FUNCTION_BLOCK FlushingManagerEffluent (* Basic Function Block Type *)
  (* Standard: 61499-2 *)
  (* Version 0.0, 8/23/2024, SESA713705, Schneider Electric, Template *)
  PACKAGE SE.Nereda;
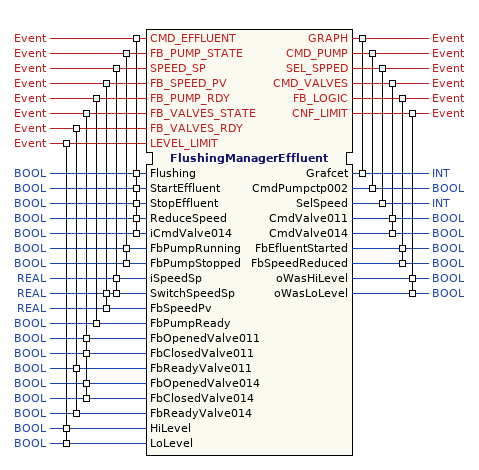
  EVENT_INPUT
    CMD_EFFLUENT WITH StartEffluent, StopEffluent, ReduceSpeed, iCmdValve014, Flushing;
    FB_PUMP_STATE WITH FbPumpRunning, FbPumpStopped;
    SPEED_SP WITH SwitchSpeedSp, iSpeedSp;
    FB_SPEED_PV WITH FbSpeedPv, SwitchSpeedSp;
    FB_PUMP_RDY WITH FbPumpReady;
    FB_VALVES_STATE WITH FbOpenedValve014, FbClosedValve014, FbOpenedValve011, FbClosedValve011;
    FB_VALVES_RDY WITH FbReadyValve011, FbReadyValve014;
    LEVEL_LIMIT WITH HiLevel, LoLevel;
  END_EVENT
  EVENT_OUTPUT
    GRAPH WITH Grafcet;
    CMD_PUMP WITH CmdPumpctp002;
    SEL_SPPED WITH SelSpeed;
    CMD_VALVES WITH CmdValve011, CmdValve014;
    FB_LOGIC WITH FbEfluentStarted, FbSpeedReduced;
    CNF_LIMIT WITH oWasHiLevel, oWasLoLevel;
  END_EVENT
  VAR_INPUT
    Flushing : BOOL;
    StartEffluent : BOOL;
    StopEffluent : BOOL;
    ReduceSpeed : BOOL;
    iCmdValve014 : BOOL;
    FbPumpRunning : BOOL;
    FbPumpStopped : BOOL;
    iSpeedSp : REAL;
    SwitchSpeedSp : REAL;
    FbSpeedPv : REAL;
    FbPumpReady : BOOL;
    FbOpenedValve011 : BOOL;
    FbClosedValve011 : BOOL;
    FbReadyValve011 : BOOL;
    FbOpenedValve014 : BOOL;
    FbClosedValve014 : BOOL;
    FbReadyValve014 : BOOL;
    HiLevel : BOOL;
    LoLevel : BOOL;
  END_VAR
  VAR_OUTPUT
    Grafcet : INT;
    CmdPumpctp002 : BOOL;
    SelSpeed : INT;
    CmdValve011 : BOOL;
    CmdValve014 : BOOL;
    FbEfluentStarted : BOOL;
    FbSpeedReduced : BOOL;
    oWasHiLevel : BOOL;
    oWasLoLevel : BOOL;
  END_VAR
  VAR
    InGSInstaActive : BOOL;
    InGSsActive : BOOL;
    InSLBActive : BOOL;
    WasHiLevel : BOOL := FALSE;
    WasLoLevel : BOOL := TRUE;
  END_VAR
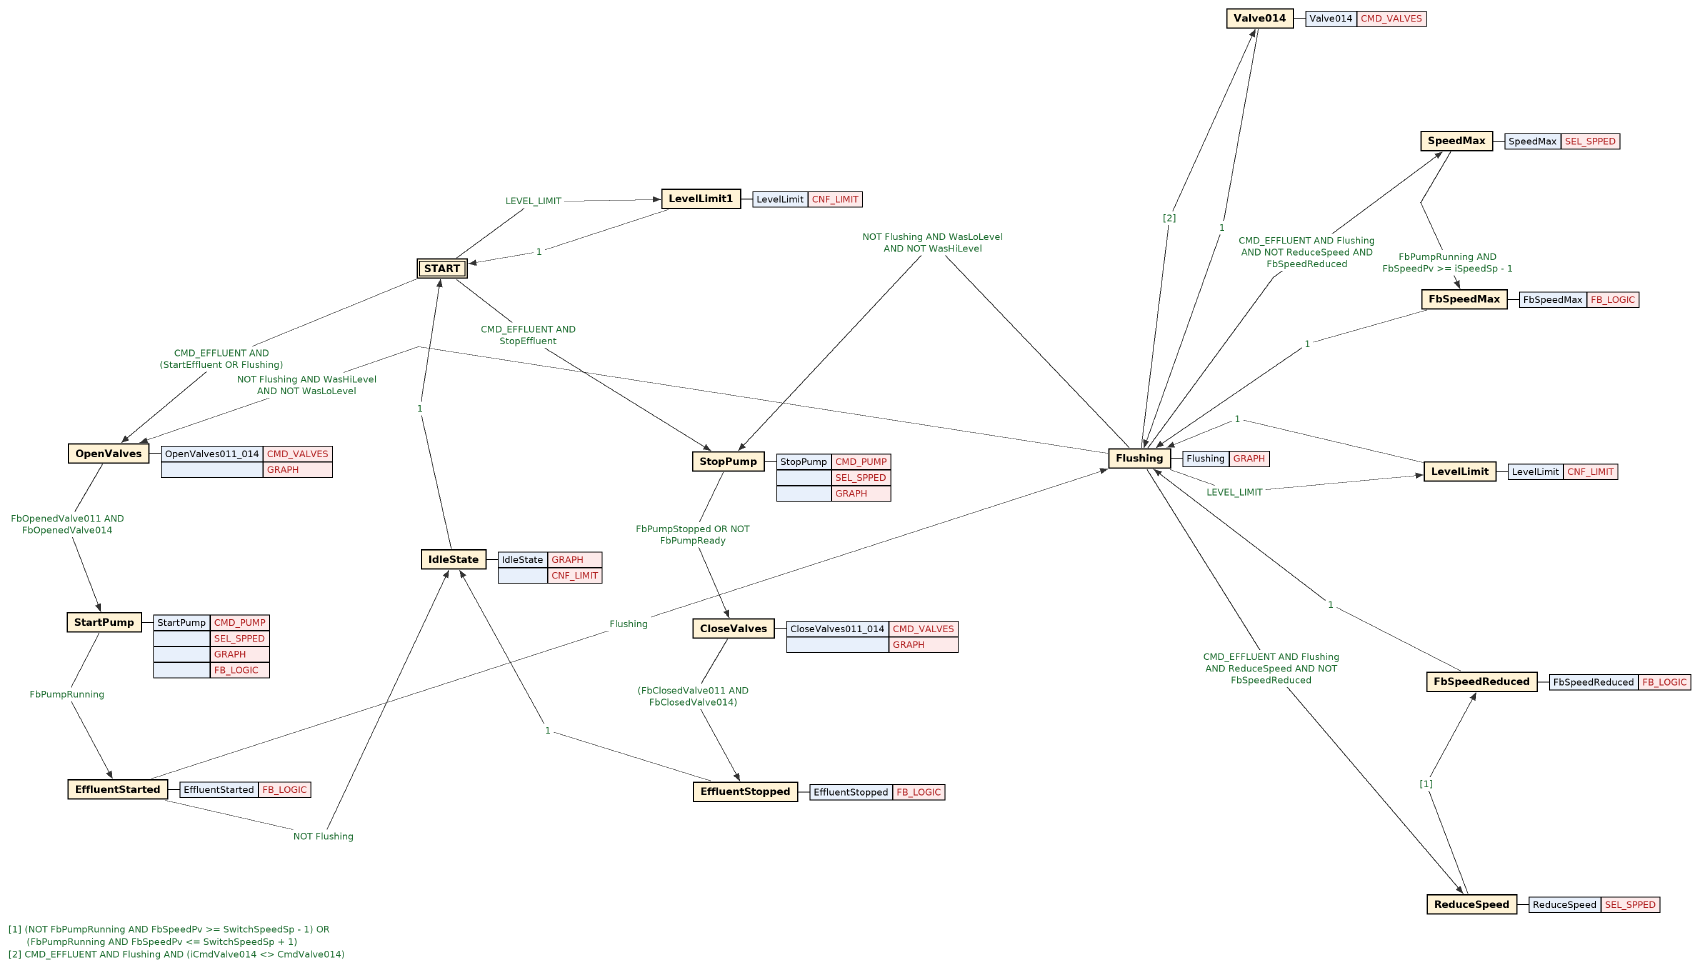
  EC_STATES
    START; (* Initial State *)
    OpenValves : OpenValves011_014 -> CMD_VALVES, -> GRAPH;
    StartPump : StartPump -> CMD_PUMP, -> SEL_SPPED, -> GRAPH, -> FB_LOGIC;
    StopPump : StopPump -> CMD_PUMP, -> SEL_SPPED, -> GRAPH;
    CloseValves : CloseValves011_014 -> CMD_VALVES, -> GRAPH;
    IdleState : IdleState -> GRAPH, -> CNF_LIMIT;
    ReduceSpeed : ReduceSpeed -> SEL_SPPED;
    SpeedMax : SpeedMax -> SEL_SPPED;
    EffluentStarted : EffluentStarted -> FB_LOGIC;
    EffluentStopped : EffluentStopped -> FB_LOGIC;
    FbSpeedMax : FbSpeedMax -> FB_LOGIC;
    FbSpeedReduced : FbSpeedReduced -> FB_LOGIC;
    Valve014 : Valve014 -> CMD_VALVES;
    Flushing : Flushing -> GRAPH;
    LevelLimit : LevelLimit -> CNF_LIMIT;
    LevelLimit1 : LevelLimit -> CNF_LIMIT;
  END_STATES
  EC_TRANSITIONS
    START TO StopPump := CMD_EFFLUENT AND StopEffluent;
    START TO OpenValves := CMD_EFFLUENT AND (StartEffluent OR Flushing);
    OpenValves TO StartPump := FbOpenedValve011 AND FbOpenedValve014;
    EffluentStarted TO IdleState := NOT Flushing;
    StopPump TO CloseValves := FbPumpStopped OR NOT FbPumpReady;
    IdleState TO START := 1;
    Flushing TO StopPump := NOT Flushing AND WasLoLevel AND NOT WasHiLevel;
    Flushing TO ReduceSpeed := CMD_EFFLUENT AND Flushing AND ReduceSpeed AND NOT FbSpeedReduced;
    FbSpeedReduced TO Flushing := 1;
    Flushing TO SpeedMax := CMD_EFFLUENT AND Flushing AND NOT ReduceSpeed AND FbSpeedReduced;
    FbSpeedMax TO Flushing := 1;
    StartPump TO EffluentStarted := FbPumpRunning;
    CloseValves TO EffluentStopped := (FbClosedValve011 AND FbClosedValve014);
    SpeedMax TO FbSpeedMax := FbPumpRunning AND FbSpeedPv >= iSpeedSp - 1;
    ReduceSpeed TO FbSpeedReduced := (NOT FbPumpRunning AND FbSpeedPv >= SwitchSpeedSp - 1) OR (FbPumpRunning AND FbSpeedPv <= SwitchSpeedSp + 1);
    Flushing TO Valve014 := CMD_EFFLUENT AND Flushing AND (iCmdValve014 <> CmdValve014);
    Valve014 TO Flushing := 1;
    EffluentStarted TO Flushing := Flushing;
    Flushing TO OpenValves := NOT Flushing AND WasHiLevel AND NOT WasLoLevel;
    Flushing TO LevelLimit := LEVEL_LIMIT;
    LevelLimit TO Flushing := 1;
    EffluentStopped TO IdleState := 1;
    START TO LevelLimit1 := LEVEL_LIMIT;
    LevelLimit1 TO START := 1;
  END_TRANSITIONS
  ALGORITHM OpenValves011_014 IN ST:
;
CmdValve011 := TRUE;
CmdValve014 := TRUE;

Grafcet := 1;
  END_ALGORITHM
  ALGORITHM StartPump IN ST:
;
CmdPumpctp002 := TRUE;
SelSpeed := 2; //Max Speed
FbSpeedReduced := FALSE;
Grafcet := 2;
  END_ALGORITHM
  ALGORITHM StopPump IN ST:
;
CmdPumpctp002 := FALSE;
SelSpeed := 0;//Speed zero

Grafcet := 3;
  END_ALGORITHM
  ALGORITHM CloseValves011_014 IN ST:
;
CmdValve011 := FALSE;
CmdValve014 := FALSE;

Grafcet := 4;
  END_ALGORITHM
  ALGORITHM IdleState IN ST:
;
Grafcet := 14;
oWasLoLevel := WasLoLevel;
oWasHiLevel := WasHiLevel;
  END_ALGORITHM
  ALGORITHM SpeedCmd IN ST:

  END_ALGORITHM
  ALGORITHM ReduceSpeed IN ST:
;
SelSpeed := 1; //Reduce Speed
  END_ALGORITHM
  ALGORITHM SpeedMax IN ST:
;
SelSpeed := 2; //Speed Max
  END_ALGORITHM
  ALGORITHM EffluentStarted IN ST:
;
FbEfluentStarted := TRUE;
FbSpeedReduced := FALSE;
  END_ALGORITHM
  ALGORITHM EffluentStopped IN ST:
;
FbEfluentStarted := FALSE;
FbSpeedReduced := TRUE;
  END_ALGORITHM
  ALGORITHM FbSpeedMax IN ST:
;
FbSpeedReduced := FALSE;
  END_ALGORITHM
  ALGORITHM FbSpeedReduced IN ST:
;
FbSpeedReduced := TRUE;
  END_ALGORITHM
  ALGORITHM Valve014 IN ST:
;
CmdValve014 := iCmdValve014;
  END_ALGORITHM
  ALGORITHM Flushing IN ST:
;
Grafcet := 15;
  END_ALGORITHM
  ALGORITHM LevelLimit IN ST:
;
IF LoLevel THEN
	WasLoLevel := TRUE;
	WasHiLevel := FALSE;
END_IF;
IF HiLevel THEN
	WasLoLevel := FALSE;
	WasHiLevel := TRUE;
END_IF;

oWasLoLevel := WasLoLevel;
oWasHiLevel := WasHiLevel;
  END_ALGORITHM
END_FUNCTION_BLOCK
